Staubli VAL3: Txt_initData.pgx

program Txt_initData()
begin
  while size(sString)>1
    $ddel(sString,size(sString)-1)
  endWhile
  while size(pfrmCad)>1
    $ddel(pfrmCad,size(pfrmCad)-1)
  endWhile
  sString[0]=""
  pfrmCad[0].trsf={0,0,0,0,0,0}
  for l_nInit=1 to 1499
    $dins(sString,l_nInit)
    $dins(pfrmCad,l_nInit)
  endFor
end
